VAR_GLOBAL
	NextfreeOrderID : INT;
	AktuellesStockwerk : INT;
	AktuellePosmm : LREAL;
	AutomatikmodusAktiv : BOOL;
	ManuellmodusAktiv : BOOL;
	AlleTuerenZu : BOOL;
	AchseSicher : BOOL;
	Fehler : ST_Error;
	Fehlertext : STRING(500);
END_VAR

(* stored: Version 1.1.0.1
   GVL Divers: Id {2fe0a1d8-72a4-4413-84d3-4a8cd0c3527c} *)
